# EPICS autosave request: stdApp/Db/ramp_tweak_settings.req
$(P)$(Q)Ramp.VAL
$(P)$(Q)TweakVal.VAL
$(P)$(Q)PutLinkCalc.AA
$(P)$(Q)RampCheckOutput.ODLY
$(P)$(Q)Ramp.OROC
